FUNCTION_BLOCK FB_Dummy
VAR_INPUT
END_VAR
VAR_OUTPUT
END_VAR
VAR
	(* not persistent variables ... *)
	iCounter		: UDINT;			(* non persistent counter *)
END_VAR
VAR PERSISTENT
	(* persistent variables ... *)
	iCounter_P		: UDINT;			(* persistent counter *)
END_VAR

iCounter 	:= iCounter + 1;
iCounter_P	:= iCounter_P + 1;

END_FUNCTION_BLOCK

(* stored: Version 1.1.0.1, ProductVersion 3.1.4024.6
   POU FB_Dummy: Id {37911085-6bab-497f-b26d-a7b12a14f0b2}, SpecialFunc None *)
